PROGRAM MAIN
VAR
END_VAR

POU();

END_PROGRAM

(* stored: Version 1.1.0.1, ProductVersion 3.1.4022.7
   POU MAIN: Id {cdd4a4f5-d3aa-47fb-9d13-ba3bf42f0f39}, SpecialFunc None *)
